GLOBALCONSTANTS FIELDBUS_SIGNAL (* Certain Constants especially for valid, error and not available *)
  (* Standard: SAE J1939; ISO 11783; Description: Copyright (c) 2023 HR Agrartechnik GmbH This program and the accompanying materials are made available under the terms of the Eclipse Public License 2.0 which is available at https://www.eclipse.org/legal/epl-2.0/ SPDX-License-Identifier: EPL-2.0 *)
  (* Version 3.1, 2026-06-01, Franz Höpfinger, HR Agrartechnik GmbH *)
  (* Version 3.0, 2025-04-14, Patrick Aigner, changed package *)
  (* Version 1.0, 2023-06-06, Franz Höpfinger, HR Agrartechnik GmbH *)
  PACKAGE eclipse4diac::signalprocessing;
  VAR_GLOBAL CONSTANT
    REVERSE : BYTE := BYTE#16#0; (* Direction reverse (0) *)
    DISABLED : BYTE := BYTE#16#0; (* Not enabled (0) *)
    DISENGAGED : BYTE := BYTE#16#0; (* Switched off (0) *)
    FORWARD : BYTE := BYTE#16#1; (* Direction forward (1) *)
    ENABLED : BYTE := BYTE#16#1; (* Enabled (1) *)
    ENGAGED : BYTE := BYTE#16#1; (* Switched on (1) *)
    ERROR_INDI_2Bit : BYTE := BYTE#16#2; (* 2 bit error indicator (2 / 0x2) *)
    NOT_AVAILABLE_2Bit : BYTE := BYTE#16#3; (* 2 bit not available (3 / 0x3) *)
    DONT_CARE_2bit : BYTE := BYTE#16#3; (* 2 bit dont care (3 / 0x3) *)
    ERROR_INDI_3Bit : BYTE := BYTE#16#6; (* 3 bit error indicator (6 / 0x6) *)
    NOT_AVAILABLE_3Bit : BYTE := BYTE#16#7; (* 3 bit not available (7 / 0x7) *)
    DONT_CARE_3bit : BYTE := BYTE#16#7; (* 3 bit dont care (7 / 0x7) *)
    ERROR_INDI_4bit : BYTE := BYTE#16#E; (* 4 bit error indicator (14 / 0xE) *)
    NOT_AVAILABLE_4bit : BYTE := BYTE#16#F; (* 4 bit not available (15 / 0xF) *)
    DONT_CARE_4bit : BYTE := BYTE#16#F; (* 4 bit dont care (15 / 0xF) *)
    VALID_SIGNAL_B : BYTE := BYTE#16#FA; (* 8 bit valid signal: 0x00..0xFA (0..250) *)
    ERROR_INDI_B : BYTE := BYTE#16#FE; (* 8 bit error indicator (254 / 0xFE) *)
    NOT_AVAILABLE_B : BYTE := BYTE#16#FF; (* 8 bit not available (255 / 0xFF) *)
    DONT_CARE_B : BYTE := BYTE#16#FF; (* 8 bit dont care (255 / 0xFF) *)
    VALID_SIGNAL_W : WORD := WORD#16#FAFF; (* 16 bit valid signal: 0x0000..0xFAFF (0..64255) *)
    ERROR_INDI_W : WORD := WORD#16#FE00; (* 16 bit error indicator min: 0xFE00 (65024) *)
    NOT_AVAILABLE_W : WORD := WORD#16#FF00; (* 16 bit not available min: 0xFF00 (65280) *)
    ERROR_INDI_WM : WORD := WORD#16#FEFF; (* 16 bit error indicator max: 0xFEFF (65279) *)
    NOT_AVAILABLE_WM : WORD := WORD#16#FFFF; (* 16 bit not available max: 0xFFFF (65535) *)
    DONT_CARE_W : WORD := WORD#16#FFFF; (* 16 bit dont care (65535 / 0xFFFF) *)
    VALID_SIGNAL_DW : DWORD := DWORD#16#FAFFFFFF; (* 32 bit valid signal: 0x00000000..0xFAFFFFFF (0..4211081215) *)
    ERROR_INDI_DW : DWORD := DWORD#16#FE000000; (* 32 bit error indicator min: 0xFE000000 *)
    NOT_AVAILABLE_DW : DWORD := DWORD#16#FF000000; (* 32 bit not available min: 0xFF000000 *)
    ERROR_INDI_DWM : DWORD := DWORD#16#FEFFFFFF; (* 32 bit error indicator max: 0xFEFFFFFF *)
    NOT_AVAILABLE_DWM : DWORD := DWORD#16#FFFFFFFF; (* 32 bit not available max: 0xFFFFFFFF *)
    DONT_CARE_DW : DWORD := DWORD#16#FFFFFFFF; (* 32 bit dont care (0xFFFFFFFF) *)
    VALID_SIGNAL_LW : LWORD := LWORD#16#FAFFFFFFFFFFFFFF; (* 64 bit valid signal: 0x0..0xFAFFFFFFFFFFFFFF (0..18086456103481911935) *)
    ERROR_INDI_LW : LWORD := LWORD#16#FE00000000000000; (* 64 bit error indicator min: 0xFE00000000000000 *)
    NOT_AVAILABLE_LW : LWORD := LWORD#16#FF00000000000000; (* 64 bit not available min: 0xFF00000000000000 *)
    ERROR_INDI_LWM : LWORD := LWORD#16#FEFFFFFFFFFFFFFF; (* 64 bit error indicator max: 0xFEFFFFFFFFFFFFFF *)
    NOT_AVAILABLE_LWM : LWORD := LWORD#16#FFFFFFFFFFFFFFFF; (* 64 bit not available max: 0xFFFFFFFFFFFFFFFF *)
    DONT_CARE_LW : LWORD := LWORD#16#FFFFFFFFFFFFFFFF; (* 64 bit dont care (0xFFFFFFFFFFFFFFFF) *)
  END_VAR
END_GLOBALCONSTANTS
